// TIA Portal V19 export
TYPE "LEXCHANGETRAY_typeRoller_toLogisticsReq"
// stored: Access Published
   STRUCT
      outFeedReq : Bool;   // 请求排料
   END_STRUCT;
END_TYPE
